// TIA Portal V17 export
// export: Created 2026-04-13T11:12:42.0235095Z, ExportSetting WithDefaults, DisplayName Totally Integrated Automation Portal, DisplayVersion V17 Update 4, DisplayName TIA Portal Openness, DisplayVersion V17 Update 4, DisplayName TIA Portal Version Control Interface, DisplayVersion V17, DisplayName SINAMICS Startdrive Advanced, DisplayVersion V17, DisplayName SINAMICS Startdrive G130, G150, S120, S150, SINAMICS MV, S210, DisplayVersion V17, DisplayName SINAMICS Startdrive G110M, G120, G120C, G120D, G120P, G115D, DisplayVersion V17, DisplayName STEP 7 Professional, DisplayVersion V17 Update 4, DisplayName STEP 7 Safety, DisplayVersion V17, DisplayName WinCC Professional, DisplayVersion V17 Update 4
FUNCTION_BLOCK "脉冲模式"   // FB39, SCL
{ S7_Optimized_Access := 'TRUE' }
VERSION : 0.1
// stored: AutoNumber true, IsIECCheckEnabled false, IsRetainMemResEnabled false, MemoryReserve 100, SetENOAutomatically false, UDAEnableTagReadback false
   VAR_IN_OUT
      QD : Bool;
      ST1 : Bool;
      ST2 : Bool;
      ST3 : Bool;
   END_VAR
   VAR
      TON1 : TON_TIME;
   END_VAR
BEGIN

   (* #BT1F := DINT_TO_TIME(REAL_TO_DINT(#BT1 * 1000.0));
   #BT2F := DINT_TO_TIME(REAL_TO_DINT(#BT1 * 1000.0)) + DINT_TO_TIME(REAL_TO_DINT(#BT2 * 1000.0));
   #BT3F := DINT_TO_TIME(REAL_TO_DINT(#BT1 * 1000.0)) + DINT_TO_TIME(REAL_TO_DINT(#BT2 * 1000.0)) + DINT_TO_TIME(REAL_TO_DINT(#BT3 * 1000.0));
   #BTAF := DINT_TO_TIME(REAL_TO_DINT(#BT1 * 1000.0)) + DINT_TO_TIME(REAL_TO_DINT(#BT2 * 1000.0)) + DINT_TO_TIME(REAL_TO_DINT(#BT3 * 1000.0)) + T#20S;
   *)
   #ST1 := 0;
   #ST2 := 0;
   #ST3 := 0;
   #QD := 0;


   IF #QD  THEN
       #TON1(IN := NOT #TON1.Q,
             PT := T#50S);

       IF #TON1.ET > T#10S THEN
               #ST1 := 1;
           END_IF;

       IF #TON1.ET >T#20S THEN
           #ST2 := 1;
       END_IF;

       IF #TON1.ET >T#30S THEN
           #ST3 := 1;
       END_IF;

       IF #TON1.ET > T#40S THEN
           #QD := 0;

       END_IF;

   END_IF;
END_FUNCTION_BLOCK
